INTERFACE IEnumerable EXTENDS IObject

METHOD GetDefaultEnumerator : IEnumerator
END_METHOD

END_INTERFACE

(* stored: Version 1.1.0.1
   Itf IEnumerable: Id {0588ef28-a449-0354-0335-eef0f6bad1aa}
   Method GetDefaultEnumerator: Id {89831ea0-8c1e-0630-3848-ccf63e8a9c7d} *)
